// TIA Portal V20 export
// export: Created 2025-12-01T14:57:23.1137598Z, ExportSetting None, DisplayName Totally Integrated Automation Portal, DisplayVersion V20 Update 3, DisplayName TIA Portal Openness, DisplayVersion V20 Update 3, DisplayName TIA Portal Version Control Interface, DisplayVersion V20 Update 3, DisplayName STEP 7 Professional, DisplayVersion V20 Update 3, DisplayName STEP 7 Safety, DisplayVersion V20 Update 2, DisplayName WinCC Basic/Comfort/Advanced, DisplayVersion V20 Update 3, DisplayName WinCC Professional, DisplayVersion V20 Update 3, DisplayName WinCC Unified, DisplayVersion V20 Update 3
DATA_BLOCK "DB911_Conf_Sistema_Scanners"   // DB911
{ S7_Optimized_Access := 'FALSE' }
AUTHOR : ROUTER
NAME : 20130623
VERSION : 3.1
// stored: AutoNumber false
   VAR RETAIN
      Bucles_lectura_Scanner { S7_SetPoint := 'True'} : Array[1..5] of "ROUT_Conf_Bucle_Lect_SCR";
   END_VAR
BEGIN
END_DATA_BLOCK
